// S11: a second program-cycle OB. Program-cycle OBs run in number order, so this
// one runs after Main (OB1) in every cycle and S2's sources stay untouched.
ORGANIZATION_BLOCK "S11Cycle"
TITLE = "S11 GRAPH rig (Program cycle)"
{ S7_Optimized_Access := 'TRUE' }
VERSION : 0.1


BEGIN
	"S11Rig"();
END_ORGANIZATION_BLOCK
